Omron CX-Programmer project NewProject (CX-Programmer 9.61)

# PLC selfHolding_latching: CP1L M
; TES SELF HOLDING USING OR NO

## Global symbols (name address type ; comment)
0.00 BOOL  ; START
0.01 BOOL  ; STOP
100.00 BOOL  ; LAMPU

## Program NewProgram1 (cyclic task 0)

### Section Section1

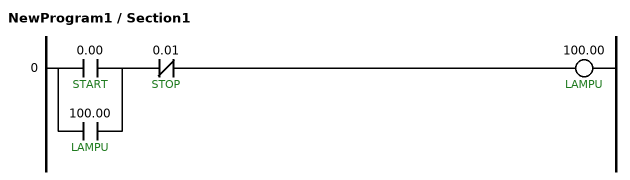
; rung 0
LD 0.00  ; START
OR 100.00  ; LAMPU
ANDNOT 0.01  ; STOP
OUT 100.00  ; LAMPU

### Section END
; rung 0
END(001)